{attribute 'enable_dynamic_creation'}
FUNCTION_BLOCK FB_TwinCATCamera EXTENDS FB_Camera
VAR
	// TwinCAT Camera specific properties
END_VAR

// TwinCAT Camera implementation

END_FUNCTION_BLOCK

(* stored: Version 1.1.0.1
   POU FB_TwinCATCamera: Id {f1b2c3d4-5556-5555-5555-555555555555} *)
